PROGRAM PRG_FactoryIO_ModbusTCP_Read
// Dépendance Tc2_ModbusSrv (TF6250-Modbus-TCP)
// FB_Bool_To_Word + FB_Word_To_Bool
VAR
	fb_FactoryIO_ModbusTCP_Read : FB_FactoryIO_ModbusTCP_Read;
END_VAR

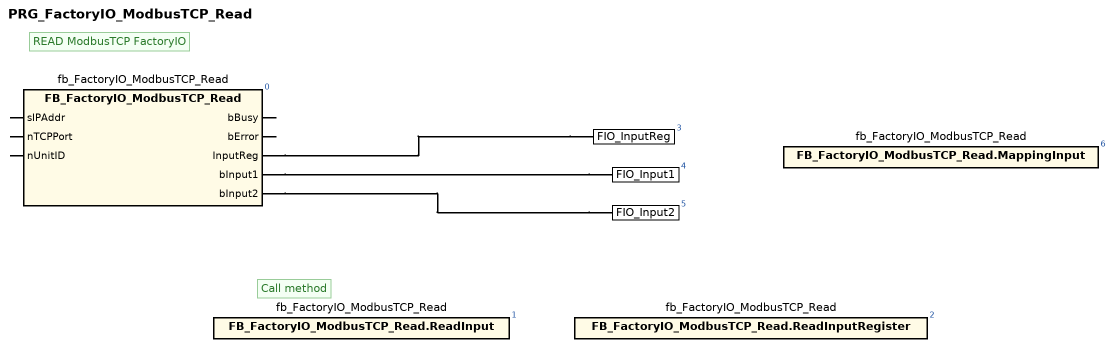
// READ ModbusTCP FactoryIO
fb_FactoryIO_ModbusTCP_Read();
// Call method
fb_FactoryIO_ModbusTCP_Read.ReadInput();
fb_FactoryIO_ModbusTCP_Read.ReadInputRegister();
FIO_InputReg := fb_FactoryIO_ModbusTCP_Read.InputReg;
FIO_Input1 := fb_FactoryIO_ModbusTCP_Read.bInput1;
FIO_Input2 := fb_FactoryIO_ModbusTCP_Read.bInput2;
fb_FactoryIO_ModbusTCP_Read.MappingInput();

END_PROGRAM

(* stored: Version 1.1.0.1, ProductVersion 3.1.4024.11
   POU PRG_FactoryIO_ModbusTCP_Read: Id {e3a0b526-1f07-43ca-9585-e7d3202c3fc5}, SpecialFunc None *)
